FUNCTION_BLOCK Sobel (* openCV sobel filter *)
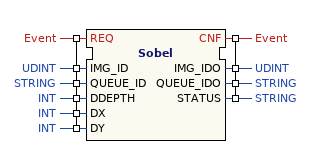
  EVENT_INPUT
    REQ WITH IMG_ID, QUEUE_ID, DDEPTH, DX, DY;
  END_EVENT
  EVENT_OUTPUT
    CNF WITH IMG_IDO, QUEUE_IDO, STATUS;
  END_EVENT
  VAR_INPUT
    IMG_ID : UDINT;
    QUEUE_ID : STRING;
    DDEPTH : INT;
    DX : INT;
    DY : INT;
  END_VAR
  VAR_OUTPUT
    IMG_IDO : UDINT;
    QUEUE_IDO : STRING;
    STATUS : STRING;
  END_VAR
END_FUNCTION_BLOCK
